// TIA Portal V20 export
// export: Created 2026-04-28T10:08:00.0471084Z, ExportSetting WithDefaults, DisplayName Totally Integrated Automation Portal, DisplayVersion V20, DisplayName TIA Portal Openness, DisplayVersion V20, DisplayName TIA Portal Version Control Interface, DisplayVersion V20, DisplayName SINAMICS Startdrive Advanced, DisplayVersion V20, DisplayName SINAMICS Startdrive G130, G150, S120, S150, SINAMICS MV, G220, S200, S210, DisplayVersion V20, DisplayName SINAMICS Startdrive G110M, G120, G120C, G120D, G120P, G115D, DisplayVersion V20, DisplayName STEP 7 Professional, DisplayVersion V20, DisplayName STEP 7 Safety, DisplayVersion V20, DisplayName WinCC Basic/Comfort/Advanced, DisplayVersion V20, DisplayName WinCC Unified, DisplayVersion V20
VAR_GLOBAL   // PLC tag table "GlobVar_PLC_IO"
   di24VDC AT %I22.4 : Bool;   // Supply 24VDC Diagnostics 24VDC
   di2WayAftCy1 AT %M0.1 : Bool;   // Rohrklappenkasten nach Zyklon 1 ES4051
   di2WayAftCy2 AT %M0.2 : Bool;   // Rohrklappenkasten nach Zyklon 2 ES4052
   di2WayBin1 AT %M0.3 : Bool;   // Rohrklappenkasten unter Zyklon 1 -> Tonne ES4012
   di2WayBin2 AT %M0.4 : Bool;   // Rohrklappenkasten unter Zyklon 2 -> Tonne ES4022
   di2WayFb1 AT %M0.5 : Bool;   // Rohrklappenkasten unter Zyklon 1 -> Rückführung ES4011
   di2WayFb2 AT %M0.6 : Bool;   // Rohrklappenkasten unter Zyklon 2 -> Rückführung ES4021
   di2WayRetCy1 AT %M0.7 : Bool;   // Rohrklappenkasten Rückführung Zyklon 1 ES4041
   di2WayRetCy2 AT %M1.0 : Bool;   // Rohrklappenkasten Rückführung Zyklon 2 ES4042
   diAckBinL AT %M1.1 : Bool;   // Quittierung Fass 2 SP3011
   diAckBinR AT %M1.2 : Bool;   // Quittierung Fass 1 SP3012
   diAgitatorOnExt_1 AT %M1.3 : Bool;   // Rührwerk 1 aus extern S6009
   diAgitatorOffExt_1 AT %M1.4 : Bool;   // Rührwerk 1 ein extern S6010
   diBuFail AT %I22.0 : Bool;   // Maxon-Brenner, Störung Maxon_Stö
   diBuFail2 AT %M1.6 : Bool;   // Maxon-Brenner 2, Störung Maxon-2_Stö
   diBuOn AT %M1.7 : Bool;   // Maxon-Brenner, Ein Maxon_Ein
   diBuOn2 AT %M2.0 : Bool;   // Maxon-Brenner 2, eingeschaltet Maxon-2_Ein
   diBuOper AT %I22.1 : Bool;   // Maxon-Brenner, in Betrieb Maxon_Betr
   diBuOper2 AT %M2.2 : Bool;   // Maxon-Brenner 2, in Betrieb Maxon-2_Betr
   diCompAir AT %I23.0 : Bool;   // Druckluft Filter ES5006
   diEmOff AT %M2.4 : Bool;   // Not - Aus NA_PNOZ
   diFillBinL AT %M2.5 : Bool;   // Abfüllanlage Befüllung Fass 1 ES3011
   diFillBinR AT %M2.6 : Bool;   // Abfüllanlage Befüllung Fass 2 ES3012
   diFlyFB_1 AT %M2.7 : Bool;   // Funkenflugüberwachung Störung #1 Funkenfl_Stö_1
   diFlyFB_10 AT %M3.0 : Bool;   // Funkenflugüberwachung Warnung #10 Funkenfl_Warn
   diFlyFB_4 AT %M3.1 : Bool;   // Funkenflugüberwachung Störung #4 Funkenfl_Stö_4
   diFuAgitator_1 AT %M3.2 : Bool;   // Rührwerk 1 Störung FU M6052_Stö_FU
   diFuDeliFan AT %M3.3 : Bool;   // Schiebeventilator Störung FU M1050_Stö_FU
   diFuMainFa AT %M3.4 : Bool;   // Hauptventilator Störung FU M5050_Stö_FU
   diFuPrede AT %M3.5 : Bool;   // Staubförderventilator Störung FU M4050_Stö_FU
   diFuSlPump1 AT %M3.6 : Bool;   // Schlickerpumpe 1 Störung FU M6050_Stö_FU
   diFuSlPump2 AT %M3.7 : Bool;   // Schlickerpumpe 2 Störung FU M6051_Stö_FU
   diGasRate AT %M4.0 : Bool;   // Gasmenge B1004
   diGrGate1 AT %M4.1 : Bool;   // Granulatweiche Stellung 1 B3008/1
   diGrGate2 AT %M4.2 : Bool;   // Granulatweiche Stellung 2 B3008/2
   diMemBreak AT %I23.4 : Bool;   // Membranbruch 1 ES6001
   diMemBreak2 AT %I23.5 : Bool;   // Membranbruch 2 ES6002
   diMpAgitator_1 AT %M4.5 : Bool;   // Motorschutz Rührwerk 1 M6052_MS
   diMpCoBe AT %M4.6 : Bool;   // Motorschutz Förderband M3051_MS
   diMpDeliFan AT %M4.7 : Bool;   // Motorschutz Schiebeventilator M1050_MS
   diMpMainFa AT %M5.0 : Bool;   // Motorschutz Hauptventilator M5050_MS
   diMpPrede AT %I22.2 : Bool;   // Motorschutz Staubförderventilator M4050_MS
   diMpRid AT %M5.2 : Bool;   // Motorschutz Rüttelsieb M3050_MS
   diMpRotFe AT %I23.2 : Bool;   // Motorschutz Zellenradschleuse Zyklon M4052_MS
   diMpSlPump AT %I23.3 : Bool;   // Motorschutz Schlickerpumpe 1 M6050_MS
   diMpSlPump2 AT %M5.5 : Bool;   // Motorschutz Schlickerpumpe 2 M6051_MS
   diMpViCo1 AT %M5.6 : Bool;   // Motorschutz Vibrationsrinne 1 M3052_MS
   diMpViCo2 AT %M5.7 : Bool;   // Motorschutz Vibrationsrinne 2 M3053_MS
   diRetHo1 AT %M6.0 : Bool;   // Staubrückführschlauch 1 ES4031
   diRetHo2 AT %M6.1 : Bool;   // Staubrückführschlauch 2 ES4032
   diSlPuOffExt AT %M6.2 : Bool;   // Schlickerpumpe aus extern S6006
   diSlPuOnExt AT %M6.3 : Bool;   // Schlickerpumpe ein extern S6005
   diSlSuppOffExt AT %M6.4 : Bool;   // Schlickerzuführung aus extern S6008
   diSlSuppOnExt AT %M6.5 : Bool;   // Schlickerzuführung ein extern S6007
   diTwPeVaBotCl AT %M6.6 : Bool;   // Doppelpendelklappe unten geschlossen ES3016
   diTwPeVaBotOp AT %M6.7 : Bool;   // Doppelpendelklappe unten geöffnet ES3015
   diTwPeVaTopCl AT %M7.0 : Bool;   // Doppelpendelklappe oben geschlossen ES3014
   diTwPeVaTopOp AT %M7.1 : Bool;   // Doppelpendelklappe oben geöffnet ES3013
   diEmOff_60 AT %M7.2 : Bool;   // Not - Aus (Schlickerversorgung) NA_PNOZ
   diEmOff_10 AT %M7.3 : Bool;   // Not - Aus (Heißluftleitung) NA_PNOZ
   diEmOff_30 AT %M7.4 : Bool;   // Not - Aus (Austrag) NA_PNOZ
   diVibLimitSw_40 AT %M7.5 : Bool;   // Vibrationsgrenzschalter, Füllstand Vorentstaubung ES4060
   diCleanDoor AT %M7.6 : Bool;   // Reinigungstür Überwachung ES2001
   diVibLimitSw_50 AT %M7.7 : Bool;   // Vibrationsgrenzschalter, Füllstand Nachentstaubung ES5060
   diMpAgitator_2 AT %M8.0 : Bool;   // Motorschutz Rührwerk 2 M6053_MS
   diFuAgitator_2 AT %M8.1 : Bool;   // Rührwerk 2 Störung FU M6053_Stö_FU
   diMpAgitator_3 AT %M8.2 : Bool;   // Motorschutz Rührwerk 3 M6054_MS
   diFuAgitator_3 AT %M8.3 : Bool;   // Rührwerk 3 Störung FU M6054_Stö_FU
   diMpAgitator_4 AT %M8.4 : Bool;   // Motorschutz Rührwerk 4 M6055_MS
   diFuAgitator_4 AT %M8.5 : Bool;   // Rührwerk 4 Störung FU M6055_Stö_FU
   diAgitatorOnExt_2 AT %M8.6 : Bool;   // Rührwerk 2 ein extern S6011
   diAgitatorOffExt_2 AT %M8.7 : Bool;   // Rührwerk 2 aus extern S6012
   diAgitatorOnExt_3 AT %M9.0 : Bool;   // Rührwerk 3 ein extern S6013
   diAgitatorOffExt_3 AT %M9.1 : Bool;   // Rührwerk 3 aus extern S6014
   diAgitatorOnExt_4 AT %M9.2 : Bool;   // Rührwerk 4 ein extern S6015
   diAgitatorOffExt_4 AT %M9.3 : Bool;   // Rührwerk 4 aus extern S6016
   diExternSignal_1 AT %M9.4 : Bool;   // Signal 1 extern, Freigabe
   diSlSupp_Water AT %M9.5 : Bool;   // Endstellung Di-Wasser, Ventil Schlickerzuführung ES
   diSlSupp_Slip AT %M9.6 : Bool;   // Endstellung Schlicker, Ventil Schlickerzuführung ES
   diMpFeedWorm AT %M9.7 : Bool;   // Motorschutz Förderschnecke
   diManPrede AT %M10.0 : Bool;   // Staubförderventilator Handfunktion FU M43S4
   diMSCombAirFan AT %M10.1 : Bool;   // Motorschutz Verbrennungsluft Geblaese
   diHoAiTeTB45 AT %M10.2 : Bool;   // Heissluftüberwachung TB45 Ausgelöst
   diExAiTeTB45 AT %M10.3 : Bool;   // Abluftüberwachung TB45 Ausgelöst
   diPrAi AT %M10.4 : Bool;   // Dungsschalter
   diFillLimitSw_2 AT %M10.5 : Bool;   // Abfüllanlage Befüllung Fass 2
   diFillLimitSw_1 AT %M10.6 : Bool;   // Abfüllanlage Befüllung Fass 1
   diMainFanSpReady AT %M10.7 : Bool;   // Option Hauptventilator mit Spülung,Fertig
   diMpWtPuDeDust AT %M11.0 : Bool;   // Motorschutz Wasserpumpe Nassentstaubung
   diMpCoBe_2 AT %M11.1 : Bool;   // Motorschutz Förderband 2
   diTeCaFail AT %M11.2 : Bool;   // Temperaturüberwachung Schaltschrank Störung
   diCoBe_2_Rev_HK AT %M11.3 : Bool;   // Förderband 2 Reversieren Hardware Schalter
   diFillBin01 AT %M11.4 : Bool;   // Abfüllanlage Befüllung Fass 1 Schalter 52S2 Kundenspezifisch
   diFillBin02 AT %M11.5 : Bool;   // Abfüllanlage Befüllung Fass 2 Schalter 52S2 Kundenspezifisch
   diFillBin03 AT %M11.6 : Bool;   // Abfüllanlage Befüllung Fass 3 Schalter 52S2 Kundenspezifisch
   diFillBin04 AT %M11.7 : Bool;   // Abfüllanlage Befüllung Fass 4 Schalter 52S2 Kundenspezifisch
   diFillBin05 AT %M12.0 : Bool;   // Abfüllanlage Befüllung Fass 5 Schalter 52S2 Kundenspezifisch
   diSwMaint AT %M12.1 : Bool;   // Schlüsselschalter für Wartung Schalter 32S7.2 Kundenspezifisch
   diSwLaTest AT %M12.2 : Bool;   // Lampentest Schalter 33SP2 Kundenspezifisch
   diBuBuStart AT %M12.3 : Bool;   // Start Taster für Brenner 34SP2 Kundenspezifisch
   diBuBuStop AT %M12.4 : Bool;   // Stop Taster für Brenner 34S4 Kundenspezifisch
   diBuSlStart AT %M12.5 : Bool;   // Start Taster für Schlickerpumpe 34SP5 Kundenspezifisch
   diBuSlStop AT %M12.6 : Bool;   // Stop Taster für Schlickerpumpe 34S7 Kundenspezifisch
   diBuFaAckn AT %M12.7 : Bool;   // Störung Quittieren 34S9 Kundenspezifisch
   diTeCaFail_2 AT %M13.0 : Bool;   // Temperaturüberwachung Schaltschrank 2 Störung
   diCleanFlapOp AT %M13.1 : Bool;   // Reinigungsklappe geöffnet
   diCleanFlapCl AT %M13.2 : Bool;   // Reinigungsklappe geschlossen
   diCleanExReq AT %M13.3 : Bool;   // Reinigungseinheit Anforderderung Reinigen
   diCleanExFin AT %M13.4 : Bool;   // Reinigungseinheit beendet
   diFiFail AT %M13.5 : Bool;   // Filtersystem keine Störmeldung
   diFiOverTemp AT %M13.6 : Bool;   // Filtersystem Übertemperatur
   diFiAlarmTemp AT %M13.7 : Bool;   // Filtersystem Alarm Temperatur
   diCleanExFail AT %M14.0 : Bool;   // Reinigungseinheit Störung
   diCleanExActiv AT %M14.1 : Bool;   // Reinigungseinheit Aktiv
   diStartEnable AT %M14.2 : Bool;   // Freigabe Start Spruehen
   diSlPuEnable AT %M14.3 : Bool;   // Freigabe Schlickerpumpe
   diLifebit AT %M14.4 : Bool;   // Lifebit
   diCleanBDEActiv AT %M14.5 : Bool;   // Reinigungseinheit BDE Aktiv
   diCleanBDEFin AT %M14.6 : Bool;   // Reinigungseinheit BDE beendet
   diExtSlEmpty AT %M14.7 : Bool;   // Externe Signal Schlicker Vorrat leer
   diCtrlCoBe1_1 AT %M15.0 : Bool;   // Überwachung Förderband 1 B3051
   diCtrlCoBe1_2 AT %M15.1 : Bool;   // Überwachung Förderband 2 B3052
   diMainFanFlapFail AT %M15.2 : Bool;   // Klappesteuerung Hauptventilator Störung
   diCyFillingMax AT %M15.3 : Bool;   // Zyklon Behälter Füllstand Max B4003
   diBinLevelMax AT %M15.4 : Bool;   // Füllstand Pufferbehälter Max B3010
   diUeberCOverflow AT %M15.5 : Bool;   // Überkorn Behälter Voll
   diEHLimFail AT %M15.6 : Bool;   // Elektroheizung Störung Begrenzer, Störung Extern
   diEHTempFail AT %M15.7 : Bool;   // Elektroheizung Störung Temperartutüberwachung, Störung Extern
   diEHAirFail AT %M16.0 : Bool;   // Elektroheizung Störung Luftströmung, Störung Extern
   diEHThy1Fail AT %M16.1 : Bool;   // Elektroheizung Störung Thyristor 1, Störung Extern
   diEHThy2Fail AT %M16.2 : Bool;   // Elektroheizung Störung Thyristor 2, Störung Extern
   diHoAiTeEHTB45 AT %M16.3 : Bool;   // Heissluftüberwachung Elektroheizung TB45 Ausgelöst
   diPrAi_Fail AT %M16.4 : Bool;   // Dungsschalter Störmeldung
   diStillstand_ZSS AT %M16.5 : Bool;   // Meldung Stillstand Zerstäuberscheibe
   diSWErreicht_ZSS AT %M16.6 : Bool;   // Meldung Sollwert erreicht Zerstäuberscheibe
   diBetriebsbereit_ZSS AT %M16.7 : Bool;   // Relais Betriebsbereit Zerstäuberscheibe
   do2WayAftCy1a AT %M20.0 : Bool;   // Rohrklappen nach Zyklon 1a PY4051
   do2WayAftCy1b AT %M20.1 : Bool;   // Rohrklappen nach Zyklon 1b PY4052
   do2WayDuRe1 AT %M20.2 : Bool;   // Rohrklappenkasten Rückführung 1 PY4041
   do2WayDuRe2 AT %M20.3 : Bool;   // Rohrklappenkasten Rückführung 2 PY4042
   do2WayUnCy1a AT %M20.4 : Bool;   // Rohrklappen unter Zyklon 1a PY4011
   do2WayUnCy1b AT %M20.5 : Bool;   // Rohrklappen unter Zyklon 1b PY4012
   do2WayUnCy2a AT %M20.6 : Bool;   // Rohrklappen unter Zyklon 2a PY4021
   do2WayUnCy2b AT %M20.7 : Bool;   // Rohrklappen unter Zyklon 2b PY4022
   doAgitator_1 AT %M21.0 : Bool;   // Rührwerk 1 Aus/Ein M6052_A/E
   doBinL AT %M21.1 : Bool;   // Fass links, Leuchte SP3011
   doBinR AT %M21.2 : Bool;   // Fass rechts, Leuchte SP3012
   doBuAck AT %Q22.6 : Bool;   // Maxon-Brenner, Quittieren Maxon_Quit
   doBuDown AT %M21.4 : Bool;   // Maxon-Brenner, Brenner Kühlen Maxon_Kühlen
   doBuEnab AT %Q22.5 : Bool;   // Maxon-Brenner, Freigabe Maxon_Freig
   doBuUp AT %M21.6 : Bool;   // Maxon-Brenner, Brenner Heizen Maxon_Heizen
   doCoBe AT %M21.7 : Bool;   // Förderband Aus/Ein M3051_A/E
   doDeliFan AT %M22.0 : Bool;   // Schiebeventilator Aus/Ein M1050_A/E
   doExAiTe AT %M22.1 : Bool;   // Abluftemperaturregelung ein Abluft_Temp_Reg
   doFailHo AT %Q22.1 : Bool;   // Sprühtrockner Störung Hupe MFL_Hupe
   doFailRed AT %Q22.2 : Bool;   // Sprühtrockner Störung rot MFL_Stö
   doFailYe AT %Q22.3 : Bool;   // Sprühtrockner Vorwarnung gelb MFL_Vorw
   doFiSy AT %Q23.3 : Bool;   // Filtersystem ein ES5009
   doFlySp AT %M22.6 : Bool;   // Funkenflugüberwachung Freigabe Funkenfl_Freig
   doFreshAir AT %Q23.2 : Bool;   // Frischluftklappe PY5001
   doKnVa2010 AT %Q24.0 : Bool;   // Klopfventil 2010 PY2010
   doKnVa2011 AT %Q24.1 : Bool;   // Klopfventil 2011 PY2011
   doKnVa2012 AT %Q24.2 : Bool;   // Klopfventil 2012 PY2012
   doKnVa2110 AT %M23.3 : Bool;   // Klopfventil 2110 PY2110
   doKnVa2111 AT %M23.4 : Bool;   // Klopfventil 2111 PY2111
   doKnVa2112 AT %M23.5 : Bool;   // Klopfventil 2112 PY2112
   doKnVa4061 AT %M23.6 : Bool;   // Klopfventil 4061, am Zyklon 1 PY4061
   doKnVa4062 AT %M23.7 : Bool;   // Klopfventil 4062, am Zyklon 2 PY4062
   doMainFaDelta AT %M24.0 : Bool;   // Hauptventilator (Dreieck) M5050_Dreieck
   doMainFan AT %Q23.1 : Bool;   // Hauptventilator Aus/Ein M5050_A/E
   doMainFaStar AT %M24.2 : Bool;   // Hauptventilator (Stern) M5050_Stern
   doPrede AT %M24.3 : Bool;   // Staubförderventilator Aus/Ein M4050_A/E
   doReGrHuReg AT %M24.4 : Bool;   // Restfeuchteregelung ein Restf_Reg
   doRid AT %M24.5 : Bool;   // Rüttelsieb Aus/Ein M3050_A/E
   doRotFe AT %Q23.5 : Bool;   // Zellenradschleuse Aus/Ein Zyklon M4052_A/E
   doSelBinL AT %M24.7 : Bool;   // Anwahl Fass 2 PY3011
   doSelBinR AT %M25.0 : Bool;   // Anwahl Fass 1 PY3012
   doSlPump AT %M25.1 : Bool;   // Schlickerpumpe 1 Aus/Ein M6050_A/E
   doSlPump2 AT %M25.2 : Bool;   // Schlickerpumpe 2 Aus/Ein M6051_A/E
   doSlSupp AT %M25.3 : Bool;   // Schlickerzuführung ein SB6007_TL
   doSlSuppOnOff AT %M25.4 : Bool;   // Schlickerzuführung ein/aus PY6001
   doSoftReg AT %M25.5 : Bool;   // Anwahl mit Software Regler Temp
   doSpDrLi AT %Q22.7 : Bool;   // Sprühtrockner Beleuchtung Turmbel_A/E
   doTwPeVaBotCl AT %M25.7 : Bool;   // Doppelpendelklappe unten schliessen PY3016
   doTwPeVaBotOp AT %M26.0 : Bool;   // Doppelpendelklappe unten öffnen PY3015
   doTwPeVaTopCl AT %M26.1 : Bool;   // Doppelpendelklappe oben schliessen PY3014
   doTwPeVaTopOp AT %M26.2 : Bool;   // Doppelpendelklappe oben öffnen PY3013
   doViCo1 AT %M26.3 : Bool;   // Vibrationsrinne 1 Aus/Ein M3052_A/E
   doViCo2 AT %M26.4 : Bool;   // Vibrationsrinne 2 Aus/Ein M3053_A/E
   doKnVa2210 AT %M26.5 : Bool;   // Klopfventil 2210 PY2210
   doKnVa2211 AT %M26.6 : Bool;   // Klopfventil 2211 PY2211
   doKnVa2212 AT %M26.7 : Bool;   // Klopfventil 2212 PY2212
   doKnVa5061 AT %M27.0 : Bool;   // Klopfventil 5061, am Filter 1 PY5061
   doKnVa5062 AT %M27.1 : Bool;   // Klopfventil 5062, am Filter 2 PY5062
   doAgitator_2 AT %M27.2 : Bool;   // Rührwerk 2 Aus/Ein M6053_A/E
   doAgitator_3 AT %M27.3 : Bool;   // Rührwerk 3 Aus/Ein M6054_A/E
   doAgitator_4 AT %M27.4 : Bool;   // Rührwerk 4 Aus/Ein M6055_A/E
   doSlSuppValve AT %M27.5 : Bool;   // Umschaltventil Schlickerzuführung PY6002
   doExternSignal_1 AT %M27.6 : Bool;   // Signal 1 extern, Freigabe Frisch
   doExternSignal_2 AT %M27.7 : Bool;   // Signal 2 extern, Überlauf
   doFeedWorm AT %M28.0 : Bool;   // Förderschnecke
   doBuSafetyCha1 AT %M28.1 : Bool;   // Sicherheit Stopp Kanal 1
   doBuSafetyCha2 AT %M28.2 : Bool;   // Sicherheit Stopp Kanal 2
   doCounterHour AT %M28.3 : Bool;   // Betriebsstundenzaehler
   doOmAck AT %Q22.0 : Bool;   // Quittierung für PNOZ - Reset
   doCombAirFan AT %M28.5 : Bool;   // Verbrennungsluft Geblaese
   doSlCtrlHW AT %M28.6 : Bool;   // HW Regler einschalten
   doWtPuDeDust_On AT %M28.7 : Bool;   // Motorschutz Wasserpumpe Nassentstaubung Ein / Aus
   doMpCoBe_2_On AT %M29.0 : Bool;   // Motorschutz Förderband 2 Ein / Ausschalten
   doMpCoBe_2_Rev AT %M29.1 : Bool;   // Motorschutz Förderband 2 Reversieren
   doSlPumpLi AT %M29.2 : Bool;   // Schlickerpumpe externe Lampe
   doBetriebGr AT %Q22.4 : Bool;   // Sprühtrockner Betrieb Gruen MFL_Betr
   doFailBl AT %M29.4 : Bool;   // Sprühtrockner Wartung Blau
   doLaBuBUStart AT %M29.5 : Bool;   // Lampe Start Taster für Brenner 34SP2 Kundenspezifisch
   doLaBuSlStart AT %M29.6 : Bool;   // Lampe Start Taster für Schlickerpumpe 34SP5 Kundenspezifisch
   doLaBuFaAckn AT %M29.7 : Bool;   // Lampe Störung Quittieren 34S9 Kundenspezifisch
   doCleanFlapOp AT %M30.0 : Bool;   // Reinigungsklappe öffnen
   doCleanFlapCl AT %M30.1 : Bool;   // Reinigungsklappe schliessen
   doCleanExReady AT %M30.2 : Bool;   // Sprühtrockner bereit
   doMainFanOpen AT %M30.3 : Bool;   // Abluftklappe öffnen Hauptventilator
   doMainFanClose AT %M30.4 : Bool;   // Abluftklappe Schliessen Hauptventilator
   doCleanExAckn AT %M30.5 : Bool;   // Externe Reinigung Quittierung
   doCleanExRes AT %M30.6 : Bool;   // Externe Reinigung Reserve
   doKnVa2013 AT %M30.7 : Bool;   // Klopfventil 2013 PY2013
   doFiVa5011 AT %M31.0 : Bool;   // Filterreinigung Ventil 5011 PY5011
   doFiVa5012 AT %M31.1 : Bool;   // Filterreinigung Ventil 5012 PY5012
   doFiVa5013 AT %M31.2 : Bool;   // Filterreinigung Ventil 5013 PY5013
   doFiVa5014 AT %M31.3 : Bool;   // Filterreinigung Ventil 5014 PY5014
   doFiVa5015 AT %M31.4 : Bool;   // Filterreinigung Ventil 5015 PY5015
   doFiVa5016 AT %M31.5 : Bool;   // Filterreinigung Ventil 5016 PY5016
   doMaOpActiv AT %M31.6 : Bool;   // Betriebsart Einrichten aktiv
   doAutoOpRunning AT %M31.7 : Bool;   // Betriebsart Automatik in Betrieb
   doCleanReq AT %M32.0 : Bool;   // Reinigung Anforderung
   doCleanReqFlapOp AT %M32.1 : Bool;   // Reinigungsklappe öffnen Anforderung
   doMaFailure AT %M32.2 : Bool;   // Anlage in Störung
   doLifebit AT %M32.3 : Bool;   // Lifebit
   doSlPuRunning AT %M32.4 : Bool;   // Externe Signal schlickerpumpe gestartet
   doPolyCoOn AT %M32.5 : Bool;   // Polyförderer Ein/Aus PY3017
   doPolyCoOn_2 AT %M32.6 : Bool;   // 2. Polyförderer Ein/Aus PY3018
   doProAirAvailable AT %M32.7 : Bool;   // Prozessluft Vorhanden
   doOnOff_ZSS AT %M33.0 : Bool;   // Start-Stopp Zerstäuberscheibe
   doCounterHour20 AT %M33.1 : Bool;   // Betriebsstundenzaehler D20
   doBuEnab2 AT %M33.2 : Bool;   // Maxon-Brenner, Freigabe Maxon_Freig D20
   doBuAck2 AT %M33.3 : Bool;   // Maxon-Brenner, Quittieren Maxon_Quit D20
   do_PwViVent AT %M33.4 : Bool;   // Magnetventil für Vibrationsbelüfter S02
   do_PwViMot AT %M33.5 : Bool;   // Elektrovibrator M1
   do_RotFi AT %Q23.4 : Bool;   // Zellenradschleuse Aus/Ein Filter M5052_A/E
   do_VaSwFlapOpen AT %Q23.6 : Bool;   // Ventil Umschaltung Klappe öffnen
   aiAgitator_1 AT %MW35 : Word;   // Rührwerk 1 Istwert M6052_Ist
   aiCoAi AT %IW42 : Word;   // Luftmenge Düse HB6010
   aiDeliFan AT %MW39 : Word;   // Schiebeventilator Istwert M1050_Ist
   aiDiDuFiBa AT %MW41 : Word;   // Differenzdruck Filter, Staubförderventilator HB4001
   aiDiFiBurn AT %MW43 : Word;   // Differenzdruck Brenner HB1006
   aiDiPrFi AT %IW32 : Word;   // Differenzdruck Filter HB5005
   aiDuFiMo AT %MW47 : Word;   // Staubfilter Überwachung HB5007
   aiExAiTe AT %IW48 : Word;   // Ablufttemperatur Istwert D5003
   aiFlRa AT %IW34 : Word;   // Massedurchfluss (Schlickermenge) HB6004
   aiFlRaAirBurn AT %MW53 : Word;   // Zufuhr Volumenstrom Brenner HB1007/2
   aiFlRaAirFlue AT %MW55 : Word;   // Luftvolumenstrom Kamin HB5008/1
   aiFlRaAirPrede AT %MW57 : Word;   // Luftvolumenstrom Staubrückführung HB4002/1
   aiGrTe AT %IW62 : Word;   // Granulattemperatur B3001
   aiHoAiTe AT %IW46 : Word;   // Heisslufttemperatur Istwert B1001_Ist
   aiMainFan AT %MW63 : Word;   // Hauptventilator Istwert M5050_Ist
   aiMoCu AT %MW65 : Word;   // Hauptventilator Istwert Stomaufnahme M5050_Ist_Strom
   aiPrAi AT %IW40 : Word;   // Druck Zerstäubungsluft HB6011
   aiPrCy AT %IW30 : Word;   // Unterdruck im Zyklon (Abluft) HB5003
   aiPrede AT %MW71 : Word;   // Staubförderventilator Istwert M4050_Ist
   aiPrSl AT %IW36 : Word;   // Schlickerdruck HB6003
   aiPrTo AT %IW28 : Word;   // Unterdruck im Turm HB2003
   aiReGrHu AT %MW77 : Word;   // Granulatrestfeuchte HB3002
   aiScaleL AT %MW79 : Word;   // Waage 2 Istwert HB3006
   aiScaleR AT %MW81 : Word;   // Waage 1 Istwert HB3005
   aiSlPump1 AT %MW83 : Word;   // Schlickerpumpe 1 Istwert M6050_Ist
   aiSlPump2 AT %MW85 : Word;   // Schlickerpumpe 2 Istwert M6051_Ist
   aiSlRes AT %MW89 : Word;   // Schlickervorratsbehälter HB6008
   aiSpDrTe1 AT %MW91 : Word;   // Temperatur Level 1 B2010
   aiSpDrTe2 AT %MW93 : Word;   // Temperatur Level 2 D2011
   aiSpDrTe3 AT %MW95 : Word;   // Temperatur Level 3 D2012
   aiSpDrTe4 AT %MW97 : Word;   // Temperatur Level 4 D2013
   aiTempBurn AT %MW99 : Word;   // Zufuhr Temperatur Brenner HB1007/1
   aiTempFlue AT %MW101 : Word;   // Zuführtemperatur Kamin HB5008/2
   aiTempPrede AT %MW103 : Word;   // Zuführtemperatur Staubrückführung HB4002/2
   aiDiPrSucFi AT %MW105 : Word;   // Differenzdruck Nachfilter HB5006
   aiHeatExIn AT %MW107 : Word;   // Temp. Wärmetauscher Eintritt D5010
   aiHeatExOut AT %MW109 : Word;   // Temp. Wärmetauscher Austritt D5011
   aiAgitator_2 AT %MW111 : Word;   // Rührwerk Istwert 2 M6053_Ist
   aiAgitator_3 AT %MW113 : Word;   // Rührwerk Istwert 3 M6054_Ist
   aiAgitator_4 AT %MW115 : Word;   // Rührwerk Istwert 4 M6055_Ist
   aiScaleAgitator_1 AT %MW117 : Word;   // Waage Rührwerksbehälter 1 HB6021
   aiScaleAgitator_2 AT %MW119 : Word;   // Waage Rührwerksbehälter 2 HB6022
   aiScaleAgitator_3 AT %MW121 : Word;   // Waage Rührwerksbehälter 3 HB6023
   aiScaleAgitator_4 AT %MW123 : Word;   // Waage Rührwerksbehälter 4 HB6024
   aiOelTemp AT %MW125 : Word;   // Öltemperatur Schlickerpumpe D6030
   aiTempCoolWater AT %MW127 : Word;   // Temperatur Kühlwasser B
   aiFlowCoolWater AT %MW129 : Word;   // Durchflusswächter Kühlwasser B
   aiGasRate AT %IW26 : Word;   // Gaszähler
   aiPrSl2 AT %MW133 : Word;   // Schlickerdruck 2 HB6005
   aiSlPuControl AT %MW135 : Word;   // Schlickerdruck Druckregelung
   aiViscosity1 AT %MW137 : Word;   // Viskositätsmessung 1
   aiViscosity2 AT %MW139 : Word;   // Viskositätsmessung 2
   aiTempSl AT %MW141 : Word;   // Schlickertemperatur
   aiViscoTemp AT %MW143 : Word;   // Temperatur bei der Viskositätsmessung 1
   aiLeMonitor AT %MW145 : Word;   // Füllstandsüberwachung am Pulverbehälter
   aiMainFanPosFlap AT %MW147 : Word;   // Stellglied der Klappe auf/zu
   aiFlProAir AT %IW38 : Word;   // Prozessluft Menge
   aiPrCompAir AT %MW151 : Word;   // Druckluft Filteranlage
   aiPrFiBefore AT %MW153 : Word;   // Unterdruckschalter Ansaugfilter Vor
   aiPrFiAfter AT %MW155 : Word;   // Unterdruckschalter Nach Filter
   aiFlRaCy AT %MW157 : Word;   // Strömungsüberwachung Staubrückführung HB4003
   aoAgitator_1 AT %MW159 : Word;   // Rührwerk 1 Sollwert M6052_Soll
   aoDeliFan AT %MW161 : Word;   // Schiebeventilator Sollwert M1050_Soll
   aoExAiTe AT %MW163 : Word;   // Ablufttemperatur Sollwert Abluft-Temp_Soll
   aoHoAir AT %QW30 : Word;   // Heißlufttemperatur Sollwert HL-Temp_Soll
   aoMainFan AT %MW167 : Word;   // Hauptventilator Sollwert M5050_Soll
   aoPrede AT %MW169 : Word;   // Staubförderventilator Sollwert M4050_Soll
   aoReGrHu AT %MW171 : Word;   // Restfeuchteregelung Sollwert Restfeuchte_Soll
   aoSlPump AT %MW173 : Word;   // Schlickerpumpe 1 Sollwert M6050_Soll
   aoSlPump2 AT %MW175 : Word;   // Schlickerpumpe 2 Sollwert M6051_Soll
   aoAgitator_2 AT %MW177 : Word;   // Rührwerk 2 Sollwert M6053_Soll
   aoAgitator_3 AT %MW179 : Word;   // Rührwerk 3 Sollwert M6054_Soll
   aoAgitator_4 AT %MW181 : Word;   // Rührwerk 4 Sollwert M6055_Soll
   aoLevelAgitator_1 AT %MW183 : Word;   // Istwert Füllstand Rührwerksbehälter 1
   aoLevelAgitator_2 AT %MW185 : Word;   // Istwert Füllstand Rührwerksbehälter 2
   aoLevelAgitator_3 AT %MW187 : Word;   // Istwert Füllstand Rührwerksbehälter 3
   aoLevelAgitator_4 AT %MW189 : Word;   // Istwert Füllstand Rührwerksbehälter 4
   aoSlPuControl AT %MW191 : Word;   // Schlickerdruck Druckregelung FU
   aoMainFanSetFlap AT %MW193 : Word;   // Sollwert Stellung der Klappe
   diSicherheitSchalter_ZSS AT %M17.0 : Bool;   // Sicherheitsschalter Gerät im Position
   aiIstwert_ZSS AT %MW195 : Word;   // Frequez-Istwert Zerstäuberscheibe
   aoSollwert_ZSS AT %MW197 : Word;   // Sollwert Zerstäuberscheibe
   aiTeEH_TB45 AT %MW199 : Word;   // Temperature from the electric heater via the TB45 shutdown precondition for the main fan
   aiTeEH_PwAkt AT %MW201 : Word;   // Power measurement from the electric heater Signal from the heater
   diRidOverflow AT %M17.1 : Bool;
   aiExAiTeD20 AT %MW203 : Word;   // Ablufttemperatur Istwert D5003 D20
   aiHoAiTeD20 AT %MW205 : Word;   // Heisslufttemperatur Istwert B1001_Ist D20
   aiPrCyD20 AT %MW207 : Word;   // Unterdruck im Zyklon (Abluft) HB5003 D20
   aiPrToD20 AT %MW209 : Word;   // Unterdruck im Turm HB2003 D20
   aiGasRateD20 AT %MW211 : Word;   // Gaszähler D20
   aiPrSlD20 AT %MW213 : Word;   // Schlickerdruck HB6003 D20
   aiFlRaD20 AT %MW215 : Word;   // Massedurchfluss (Schlickermenge) HB6004 D20
   diPwLeSw AT %M17.2 : Bool;   // Fuellstandsensor am Pulverzufuehrung S01
   aoHoAirD20 AT %MW217 : Word;   // Heißlufttemperatur Sollwert HL-Temp_Soll D20
   diMpRotFilter AT %I23.1 : Bool;   // Motorschutz Zellenradschleuse FilterM5052_MS
   diMemBreak3 AT %I23.6 : Bool;   // Membranbruch 3 ES6003
   diFiMonEmpty AT %I24.0 : Bool;   // Filteranlage Überwachung Niveau Sensor Leer B5060
   diFiMonFull AT %I24.1 : Bool;   // Filteranlage Überwachung Niveau Sensor Voll B5061
   diFiMonRotaryFi AT %I24.2 : Bool;   // Filteranlage Überwachung Zellenrad Filter B5062
   diFiMonRotaryCy AT %I24.3 : Bool;   // Filteranlage Überwachung Zellenrad Zyklon B4053
   doSTOPredeCh1 AT %Q0.0 : Bool;   // STO Staubförderventilator Kanal 1
   doSTOPredeCh2 AT %Q0.1 : Bool;   // STO Staubförderventilator Kanal 2
   doSTOMainFanCh1 AT %Q0.2 : Bool;   // STO Hauptventilator Kanal 1
   doSTOMainFanCh2 AT %Q0.3 : Bool;   // STO Hauptventilator Kanal 2
   doSTOSlPuCh1 AT %Q5.0 : Bool;   // STO Schlickerpumpe Kanal 1
   doSTOSlPuCh2 AT %Q5.1 : Bool;   // STO Schlickerpumpe Kanal 2
   doNHContactorCh1 AT %Q5.2 : Bool;   // Not-Halt Schütz Kanal 1
   doNHContactorCh2 AT %Q5.3 : Bool;   // Not-Halt Schütz Kanal 2
   diNHCabinetCh1 AT %I66.0 : Bool;   // Not-Halt Schaltschrank Kanal 1
   diNHSlPuCh1 AT %I66.1 : Bool;   // Not-Halt Schlickerpumpe Kanal 1
   diNHBurnerCh1 AT %I66.2 : Bool;   // Not-Halt Brenner Kanal 1
   diNHCtrlRoomCh1 AT %I66.3 : Bool;   // Not-Halt Leitwarte Kanal 1
   diNHCabinetCh2 AT %I66.4 : Bool;   // Not-Halt Schaltschrank Kanal 2
   diNHSlPuCh2 AT %I66.5 : Bool;   // Not-Halt Schlickerpumpe Kanal 2
   diNHBurnerCh2 AT %I66.6 : Bool;   // Not-Halt Brenner Kanal 2
   diNHCtrlRoomCh2 AT %I66.7 : Bool;   // Not-Halt Leitwarte Kanal 2
   diAckFail AT %I73.0 : Bool;   // Störung quittieren
   "diNHReturnCircuit Ch1Ch2" AT %I73.2 : Bool;   // Rückführkreis Not-Halt Schütz Kanal 1/2
   diNHOperPanelCh1 AT %I73.1 : Bool;   // Not-Halt Bedienpanel Kanal 1
   diBAManually AT %I73.4 : Bool;   // Betriebsart Einrichten
   diNHOperPanelCh2 AT %I73.5 : Bool;   // Not-Halt Bedienpanel Kanal 2
   diBAAutomatic AT %I73.6 : Bool;   // Betriebsart Automatik
   do_VaSwFlapClose AT %Q23.7 : Bool;   // Ventil Umschaltung Klappe schliessen
   diPreFlushActive AT %I24.4 : Bool;   // Eingang von Zeitrelais - Vorspülen aktiv!
END_VAR
